Universal Robots PolyScope program: gravityFeederW.urp

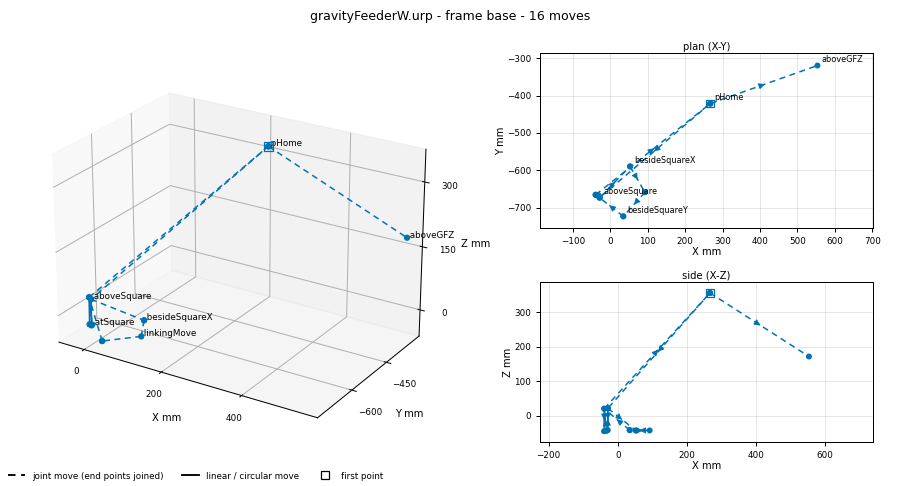
[picture p0: tool path of gravityFeederW.urp in frame base, 16 of 21 moves have a stored position in this frame; points joined in program order, loops and branches not executed]
Program gravityFeederW (installation=admin directory=/programs/WED_9AM createdIn=3.8.0.61336 lastSavedIn=3.15.8.106339 robotSerialNumber=2015350924)
Calibrated DH parameters: a=[0, -0.425, -0.39225, 0, 0, 0]; d=[0.089159, 0, 0, 0.10915, 0.09465, 0.0823]; alpha=[1.570796, 0, 0, 1.570796, -1.570796, 0]; deltaTheta=[0, 0, 0, 0, 0, 0]
Robot Program (runOnlyOnce=true)
  Set DigitalOutput pin=digital_out[0]; digitalValue=0
  Call _adminLinearIndex2
  MoveJ speed 180 deg/s, acceleration 100 deg/s^2 (useActiveTCP=true)
    Waypoint pHome: TCP in base x=267.118 y=-421.457 z=355.823 mm, rx=1.114 ry=1.1062 rz=0.0051 rad; joints [-44.998, -90.002, -90.001, -90.005, 90.001, 0.003] deg; flange x=267.125 y=-421.465 z=431.823 mm, rx=1.2022 ry=-2.9024 rz=-0.0002 rad
    Waypoint aboveGFZ: TCP in base x=553.609 y=-319.815 z=171.755 mm, rx=0.8755 ry=0.8576 rz=-0.0128 rad; joints [-17.833, -110.331, -99.527, -42.704, 80.636, 26.761] deg; flange x=536.004 y=-301.162 z=243.296 mm, rx=-1.1147 ry=2.7614 rz=-0.4822 rad
  MoveL speed 150 mm/s, acceleration 50 mm/s^2 (useActiveTCP=true) feature=Base
    Waypoint atGFRel (Relative): relativeFromPosition TCP in base x=703.737 y=-146.697 z=167.898 mm, rx=0.8752 ry=0.8574 rz=-0.0125 rad; joints [0.113, -120.689, -83.441, -52.052, 75.76, 44.404] deg; TCP in base x=721.869 y=-165.337 z=96.451 mm, rx=0.8753 ry=0.8574 rz=-0.0126 rad; joints [-1.446, -127.81, -83.304, -44.693, 76.139, 42.848] deg; flange x=704.241 y=-146.679 z=167.985 mm, rx=-1.1148 ry=2.7611 rz=-0.4824 rad
    Set DigitalOutput pin=digital_out[0]; digitalValue=1
    Wait Sleep waitTime=1
    Waypoint moveUpRel (Relative): relativeFromPosition TCP in base x=550.868 y=-331.595 z=98.44 mm, rx=0.8702 ry=0.856 rz=-0.0137 rad; joints [-18.828, -116.476, -103.566, -32.215, 80.938, 25.84] deg; TCP in base x=559.003 y=-337.636 z=101.257 mm, rx=0.8748 ry=0.8551 rz=-0.0126 rad; joints [-19.316, -117.357, -101.374, -33.468, 81.07, 25.361] deg; flange x=541.244 y=-318.91 z=172.741 mm, rx=-1.1129 ry=2.7599 rz=-0.4844 rad
    Waypoint aboveGFRel (Relative): relativeFromPosition TCP in base x=559.155 y=-339.81 z=102.554 mm, rx=0.8699 ry=0.8564 rz=-0.014 rad; joints [-19.315, -117.355, -101.372, -33.466, 81.074, 25.359] deg; TCP in base x=542.815 y=-319.749 z=167.249 mm, rx=0.8748 ry=0.8556 rz=-0.0118 rad; joints [-18.166, -109.5, -101.542, -41.339, 80.755, 26.43] deg; flange x=525.048 y=-301.069 z=238.743 mm, rx=-1.114 ry=2.7594 rz=-0.4837 rad
  MoveJ speed 180 deg/s, acceleration 100 deg/s^2 (useActiveTCP=true)
    Waypoint pHome: motionParameters(blendRadius=0.1); TCP in base x=267.118 y=-421.457 z=355.823 mm, rx=1.114 ry=1.1062 rz=0.0051 rad; joints [-44.998, -90.002, -90.001, -90.005, 90.001, 0.003] deg; flange x=267.125 y=-421.465 z=431.823 mm, rx=1.2022 ry=-2.9024 rz=-0.0002 rad
    Waypoint aboveSquare: TCP in base x=-28.511 y=-672.755 z=21.747 mm, rx=1.7065 ry=-0.0121 rz=-1.2064 rad; joints [-83.109, -128.084, -90.371, -51.361, 90.044, 52.13] deg; flange x=-28.598 y=-672.52 z=97.746 mm, rx=1.2074 ry=2.8979 rz=-0.0038 rad
  MoveL speed 250 mm/s, acceleration 1200 mm/s^2 (useActiveTCP=true) feature=Base
    Waypoint atSquare: TCP in base x=-28.895 y=-673.156 z=-41.381 mm, rx=1.7064 ry=-0.0122 rz=-1.2063 rad; joints [-83.146, -133.814, -91.573, -44.421, 90.044, 52.094] deg; flange x=-28.984 y=-672.911 z=34.619 mm, rx=1.2074 ry=2.8978 rz=-0.004 rad
    Set DigitalOutput pin=digital_out[0]; digitalValue=0
    Wait Sleep waitTime=0.5
    Waypoint aboveSquare: TCP in base x=-28.511 y=-672.755 z=21.747 mm, rx=1.7065 ry=-0.0121 rz=-1.2064 rad; joints [-83.109, -128.084, -90.371, -51.361, 90.044, 52.13] deg; flange x=-28.598 y=-672.52 z=97.746 mm, rx=1.2074 ry=2.8979 rz=-0.0038 rad
    Set DigitalOutput pin=digital_out[0]; digitalValue=1
  MoveJ speed 60 deg/s, acceleration 80 deg/s^2 (useActiveTCP=true)
    Waypoint besideSquareX: TCP in base x=52.617 y=-589.571 z=-42.423 mm, rx=1.7065 ry=-0.0117 rz=-1.2076 rad; joints [-74.267, -126.531, -106.897, -36.426, 89.974, 61.001] deg; flange x=52.598 y=-589.375 z=33.577 mm, rx=1.2085 ry=2.8985 rz=-0.0036 rad
  MoveL speed 35 mm/s, acceleration 35 mm/s^2 (useActiveTCP=true) feature=Base
    If force()≤40 (checkContinuously=true)
      Waypoint atSquareX (Relative): relativeFromPosition TCP in base x=50.865 y=-591.008 z=-41.515 mm, rx=1.7022 ry=-0.008 rz=-1.2089 rad; joints [-74.266, -126.532, -106.898, -36.426, 89.971, 60.977] deg; TCP in base x=-28.314 y=-672.475 z=-41.562 mm, rx=1.7067 ry=-0.0121 rz=-1.2064 rad; joints [-83.089, -133.766, -91.707, -44.351, 90.046, 52.151] deg; flange x=-28.404 y=-672.249 z=34.438 mm, rx=1.2075 ry=2.8979 rz=-0.0036 rad
    Wait Sleep waitTime=0.5
  MoveJ speed 60 deg/s, acceleration 80 deg/s^2 (useActiveTCP=true)
    Waypoint besideSquareX: TCP in base x=52.617 y=-589.571 z=-42.423 mm, rx=1.7065 ry=-0.0117 rz=-1.2076 rad; joints [-74.267, -126.531, -106.897, -36.426, 89.974, 61.001] deg; flange x=52.598 y=-589.375 z=33.577 mm, rx=1.2085 ry=2.8985 rz=-0.0036 rad
    Waypoint linkingMove: motionParameters(blendRadius=0.01); TCP in base x=92.406 y=-658.703 z=-42.29 mm, rx=1.7071 ry=-0.0114 rz=-1.2067 rad; joints [-72.572, -133.085, -93.255, -43.522, 90.01, 62.663] deg; flange x=92.339 y=-658.532 z=33.709 mm, rx=1.2075 ry=2.8984 rz=-0.0027 rad
    Waypoint besideSquareY: TCP in base x=34.628 y=-723.042 z=-41.53 mm, rx=1.7068 ry=-0.0118 rz=-1.2057 rad; joints [-78.597, -138.866, -81.159, -49.796, 90.051, 56.613] deg; flange x=34.515 y=-722.822 z=34.47 mm, rx=1.2066 ry=2.8979 rz=-0.0033 rad
  MoveL speed 35 mm/s, acceleration 35 mm/s^2 (useActiveTCP=true) feature=Base
    If force()≤40 (checkContinuously=true)
      Waypoint atSquareY (Relative): relativeFromPosition TCP in base x=32.384 y=-724.404 z=-40.504 mm, rx=1.7021 ry=-0.0085 rz=-1.209 rad; joints [-78.599, -138.865, -81.161, -49.795, 90.053, 56.612] deg; TCP in base x=-15.805 y=-673.754 z=-41.467 mm, rx=1.7062 ry=-0.0122 rz=-1.2065 rad; joints [-82.03, -133.837, -91.546, -44.419, 90.028, 53.212] deg; flange x=-15.879 y=-673.5 z=34.533 mm, rx=1.2075 ry=2.8979 rz=-0.0043 rad
    Wait Sleep waitTime=0.5
  MoveJ speed 60 deg/s, acceleration 80 deg/s^2 (useActiveTCP=true)
    Waypoint besideSquareY: TCP in base x=34.628 y=-723.042 z=-41.53 mm, rx=1.7068 ry=-0.0118 rz=-1.2057 rad; joints [-78.597, -138.866, -81.159, -49.796, 90.051, 56.613] deg; flange x=34.515 y=-722.822 z=34.47 mm, rx=1.2066 ry=2.8979 rz=-0.0033 rad
    Waypoint aboveSquareNew: TCP in base x=-39.171 y=-665.188 z=20.711 mm, rx=1.7064 ry=-0.0121 rz=-1.2063 rad; joints [-83.953, -127.424, -91.788, -50.601, 90.045, 51.279] deg; flange x=-39.256 y=-664.947 z=96.711 mm, rx=1.2072 ry=2.8979 rz=-0.0039 rad
    Set DigitalOutput pin=digital_out[0]; digitalValue=0
    Wait Sleep waitTime=1
  MoveL speed 250 mm/s, acceleration 1200 mm/s^2 (useActiveTCP=true) feature=Base
    Waypoint atSquareNew: TCP in base x=-39.623 y=-665.674 z=-44.47 mm, rx=1.7064 ry=-0.0122 rz=-1.2064 rad; joints [-83.996, -133.455, -92.966, -43.391, 90.044, 51.246] deg; flange x=-39.706 y=-665.432 z=31.529 mm, rx=1.2075 ry=2.8978 rz=-0.004 rad
    Set DigitalOutput pin=digital_out[0]; digitalValue=1
    Wait Sleep waitTime=1
    Waypoint easeout: TCP in base x=-32.563 y=-665.585 z=-43.483 mm, rx=1.7065 ry=-0.0122 rz=-1.2064 rad; joints [-83.384, -133.314, -93.049, -43.45, 90.044, 51.855] deg; flange x=-32.65 y=-665.346 z=32.516 mm, rx=1.2074 ry=2.8978 rz=-0.0039 rad
    Waypoint aboveSquareNew: TCP in base x=-39.171 y=-665.188 z=20.711 mm, rx=1.7064 ry=-0.0121 rz=-1.2063 rad; joints [-83.953, -127.424, -91.788, -50.601, 90.045, 51.279] deg; flange x=-39.256 y=-664.947 z=96.711 mm, rx=1.2072 ry=2.8979 rz=-0.0039 rad
  MoveJ speed 60 deg/s, acceleration 80 deg/s^2 (useActiveTCP=true)
    Waypoint pHome: TCP in base x=267.118 y=-421.457 z=355.823 mm, rx=1.114 ry=1.1062 rz=0.0051 rad; joints [-44.998, -90.002, -90.001, -90.005, 90.001, 0.003] deg; flange x=267.125 y=-421.465 z=431.823 mm, rx=1.2022 ry=-2.9024 rz=-0.0002 rad
SubProgram  [hidden by the author, left out]
SubProgram _adminLinearIndex2 [hidden by the author, left out]
